FUNCTION ASCF_GetVDWordOutputList : Word
VAR_INPUT
	Index		: INT;
END_VAR

VAR_OUTPUT
	QC			: BYTE;
	Value		: DWORD;
END_VAR

VAR_IN_OUT
	OutputList	: ARRAY[*] OF ASCF_CL_OutputType;		//Output-Element of the Adaptive Logic.
END_VAR

VAR
	tempLowerBound	: DINT;
	tempUpperBound	: DINT;
	tempResult		: WORD;
	tempUnionType	: ASCF_UnionType;				//Union type that holds only one of its possible data types at a time. The type can be selected via the "Typeselector". Independent of the selected type, every value has a quality code "VQC".
	constErrors		: ASCF_CL_EnumErrors;				//Enumeration type of the error codes of the Adaptive Logic.
	constUnionTypes	: ASCF_EnumUnionTypes;			//Enumeration type of the valid values for the "Typeselector" of a "GVR_unionType"-UDT.
END_VAR



tempResult := ASCF_GetValueOutputList(Index := Index, Value => tempUnionType, OutputList := OutputList);

IF tempResult <> constErrors.None THEN
    ASCF_GetVDWordOutputList := tempResult;
    RETURN;
END_IF;

IF tempUnionType.Typeselector <> constUnionTypes.VDWord THEN
    ASCF_GetVDWordOutputList := constErrors.TypesDoNotMatch;
    RETURN;
END_IF;

QC := tempUnionType.VQC;
Value := tempUnionType.VDWord;
ASCF_GetVDWordOutputList := constErrors.None;

END_FUNCTION

(* stored: Version 1.1.0.1, ProductVersion 3.1.4026.4
   POU ASCF_GetVDWordOutputList: Id {70780ce5-fbd4-4929-bbf6-6d2ab49eb60b}, SpecialFunc None *)
